Fanuc KAREL source: LOAD_STATUS.kl

PROGRAM T
%NOLOCKGROUP
VAR
 v0 : STRING[40]
 v1 : BOOLEAN
 v2 : BOOLEAN
BEGIN
 LOAD_STATUS(v0, v1, v2)
END T
